Fanuc KAREL source: kt00212.KL

-- PROVISIONAL review KL for V770-1; original PC SHA256 9a2e28fc4b855c2f2d5b7c11b93bbb366f3dff6698dc484e297fa5f11a06d46c
-- Incomplete behavior may be omitted. Consult companion uncertainty JSON. Do not deploy.
PROGRAM KT00212
%NOLOCKGROUP
VAR
  I2 : INTEGER
  OUT : INTEGER
-- UNRESOLVED_DECL Y1 type=002018
BEGIN
  -- UNRESOLVED_PC offsets 5-19; opcodes 2E,22,9D,33,B2
  -- UNRESOLVED_PC offsets 24-35; opcodes 2E,23
  -- UNRESOLVED_PC offsets 40-62; opcodes 22,9D,33,B1,21,46,23
  -- UNRESOLVED_PC offsets 67-71; opcodes 7F
END KT00212
